FUNCTION_BLOCK FB_CognexBarcodeScanner
VAR_INPUT
	In_bManualMode		: BOOL; // Manual Mode
	In_bAutoMode		: BOOL; // Auto Mode
	In_timeScanTimer	: TIME;
	In_iResultByte		: INT;
	In_ioDeviceFault	: BOOL;
	In_ioTriggerReady	: BOOL;
	In_ioTriggerAck		: BOOL;
	In_ioAcquiring		: BOOL;
	In_ioArrayData		: ARRAY [1..480] OF BYTE;
END_VAR
VAR_OUTPUT
	Out_bDeviceError	: BOOL;
	Out_bErrScanTimeOut : BOOL;
	Out_ioTriggerEnable	: BOOL;
	Out_ioTrigger		: BOOL;
	Out_bEnableReady	: BOOL;
	Out_bTriggerDone	: BOOL;
	Out_sAutoBarcode	: STRING;
	Out_sManualBarcode	: STRING;
	Out_GetBarcodeDone	: BOOL;	
END_VAR
VAR_IN_OUT
	InOut_bAutoTriggerEnable	: BOOL;
	InOut_bManualTriggerEnable	: BOOL;
	InOut_bAutoTrigger			: BOOL;
	InOut_bManualTrigger		: BOOL;
END_VAR
VAR
	rTrig_TriggerEnable: R_TRIG;
	fTrig_TriggerEnable: F_TRIG;
	
	rTrig_Trigger: R_TRIG;
	iStepTriggerEnable	: INT;
	iStepTrigger 		: INT;
	iforCount			: INT;
	sChar				: STRING(1);
	tonTimeOut			: TON;
	sBarcode			: STRING;
END_VAR

// Device Error
Out_bDeviceError := In_ioDeviceFault;
rTrig_TriggerEnable(CLK:=(InOut_bAutoTriggerEnable AND In_bAutoMode) OR (InOut_bManualTriggerEnable AND In_bManualMode));
fTrig_TriggerEnable(CLK:=(InOut_bAutoTriggerEnable AND In_bAutoMode) OR (InOut_bManualTriggerEnable AND In_bManualMode));
	
rTrig_Trigger(CLK:=(InOut_bAutoTrigger AND In_bAutoMode) OR (InOut_bManualTrigger AND In_bManualMode));

Out_bEnableReady := In_ioTriggerReady;

// Enable Trigger
CASE iStepTriggerEnable OF
	
	0 :
		IF rTrig_TriggerEnable.Q THEN
			Out_ioTriggerEnable := TRUE;
			iStepTriggerEnable := 10;
		ELSIF fTrig_TriggerEnable.Q THEN
			Out_ioTriggerEnable := FALSE;
			Out_bTriggerDone := FALSE;
			iStepTriggerEnable := 100;
		END_IF
		
	10:
		IF In_ioTriggerReady THEN
			InOut_bAutoTriggerEnable := TRUE;
			iStepTriggerEnable := 0;
		ELSIF fTrig_TriggerEnable.Q THEN
			Out_ioTriggerEnable := FALSE;
			Out_bTriggerDone := FALSE;
			iStepTriggerEnable := 100;
		END_IF
		
	100:
		IF NOT In_ioTriggerReady THEN
			Out_bTriggerDone := FALSE;
			iStepTriggerEnable := 0;
		END_IF
		
END_CASE

CASE iStepTrigger OF
	
	0:
		IF rTrig_Trigger.Q THEN
			Out_bErrScanTimeOut := FALSE;
			IF In_ioTriggerReady THEN
				Out_bTriggerDone := FALSE;
				Out_GetBarcodeDone := FALSE;
				Out_ioTrigger := TRUE;
				iStepTrigger := 10;
			ELSE
				Out_bTriggerDone := FALSE;
				Out_GetBarcodeDone := FALSE;
				Out_ioTriggerEnable := FALSE;
				iStepTrigger := 100;
			END_IF
		END_IF
		
	10:
		IF In_ioTriggerAck AND In_ioAcquiring THEN
			sBarcode := '';
			IF In_bAutoMode THEN
				Out_sAutoBarcode := '';
			END_IF
			IF In_bManualMode THEN
				Out_sManualBarcode := '';
			END_IF
			iStepTrigger := 20;
		END_IF
	
	20: 
		tonTimeOut(IN:= TRUE, PT:= In_timeScanTimer);
		IF NOT In_ioAcquiring THEN
			tonTimeOut(IN:= FALSE);
			FOR iforCount:=1 TO In_iResultByte BY 1 DO
				IF In_ioArrayData[iforCount] <> 0 THEN
					sChar := F_ToCHR(STRING_TO_BYTE(CONCAT('16#',WORD_TO_HEXSTR(In_ioArrayData[iforCount], 1, FALSE))));
					sBarcode:= CONCAT(sBarcode,sChar);
					IF In_bAutoMode THEN
						Out_sAutoBarcode := sBarcode;
					END_IF
					IF In_bManualMode THEN
						Out_sManualBarcode := sBarcode;
					END_IF
				END_IF
			END_FOR
			iStepTrigger := 30;
		ELSIF tonTimeOut.Q THEN
			tonTimeOut(IN:= FALSE);
			IF In_bAutoMode THEN
				InOut_bAutoTrigger := FALSE;
			END_IF
			IF In_bManualMode THEN
				InOut_bManualTrigger := FALSE;
			END_IF
			Out_bTriggerDone := TRUE;
			Out_ioTrigger := FALSE;
			Out_bErrScanTimeOut := TRUE;
			iStepTrigger := 0;
		END_IF
		
	30:	
		Out_GetBarcodeDone := TRUE;
		Out_bTriggerDone := TRUE;
		IF In_bAutoMode THEN
			InOut_bAutoTrigger := FALSE;
		END_IF
		IF In_bManualMode THEN
			InOut_bManualTrigger := FALSE;
		END_IF
		Out_ioTrigger := FALSE;
		iStepTrigger := 0;
		
	100:
		IF In_bAutoMode THEN
			InOut_bAutoTriggerEnable := TRUE;
		END_IF
		IF In_bManualMode THEN
			InOut_bManualTriggerEnable := FALSE;
		END_IF
		iStepTrigger := 110;
	
	110:
		IF In_ioTriggerReady THEN
			Out_ioTrigger := TRUE;
			iStepTrigger := 10;
		END_IF	

END_CASE

END_FUNCTION_BLOCK

(* stored: Version 1.1.0.1, ProductVersion 3.1.4024.11
   POU FB_CognexBarcodeScanner: Id {867789ec-6e41-4b02-83b2-4c05f7fdccd4}, SpecialFunc None *)
